Fanuc KAREL source: ko00024.KL

-- PROVISIONAL review KL for V770-1; original PC SHA256 7f1b47b1488e21a318078b4938de0ef95c9efe25b4bc55167b8f6063e65df571
-- Incomplete behavior may be omitted. Consult companion uncertainty JSON. Do not deploy.
PROGRAM KO00024
%NOLOCKGROUP
-- UNRESOLVED_DECL P1 type=000106
-- UNRESOLVED_DECL P2 type=000106
-- UNRESOLVED_DECL P3 type=000106
-- UNRESOLVED_DECL P4 type=000106
-- UNRESOLVED_DECL OUT type=000199
BEGIN
  -- UNRESOLVED_PC offsets 5-80; opcodes 27,27,49,7E,AD,27,49,7E,AD,27,49,7E,AD,27,49,7E,AD,76,7E,4A
  -- UNRESOLVED_PC offsets 85-89; opcodes 7F
END KO00024
